// TIA Portal V16 export
// export: Created 2020-09-21T20:06:50.079873Z, ExportSetting WithDefaults, DisplayName Totally Integrated Automation Portal, DisplayVersion V16, DisplayName TIA Portal Version Control Interface, DisplayVersion V16, DisplayName TIA Portal Openness, DisplayVersion V16, DisplayName STEP 7 Professional, DisplayVersion V16, DisplayName STEP 7 Safety, DisplayVersion V16, DisplayName WinCC Advanced, DisplayVersion V16
FUNCTION_BLOCK "FB_CM100"   // FB4, LAD
{ S7_Optimized_Access := 'TRUE' }
VERSION : 0.1
// stored: AutoNumber true, IsIECCheckEnabled false, IsRetainMemResEnabled false, MemoryReserve 100, SetENOAutomatically false, UDAEnableTagReadback false
   VAR_INPUT
      read : Bool;
      adrTag : DWord;
      length : DWord;
      hwId : HW_ANY;
      portAdr : Int;
      execute : Bool;
      tagPresent : Bool;
   END_VAR
   VAR_OUTPUT
      done : Bool;
      error : Bool;
      status : DWord;
      presence : Bool;
   END_VAR
BEGIN

REGION Network 1
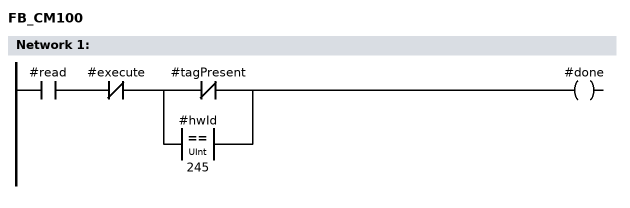
   RUNG wire#powerrail
      Contact( #read )
      I_Contact( #execute )
      wire#w1
      I_Contact( #tagPresent )
      wire#w2
      Coil( #done )
   END_RUNG
   RUNG wire#w1
      { S7_Templates := "SrcType := UInt" } EQ_Contact(in1 := #hwId, in2 := 245)
   END_RUNG wire#w2
   // the same network as SCL:
   #done := #read AND NOT #execute AND (NOT #tagPresent OR (#hwId = 245));
END_REGION
END_FUNCTION_BLOCK
